(* IEC 61131-3 sources: volt/packages/volt-lsp-iec/test-corpus/pro2193/Device/Plc Logic/Application/03 Hardware Units/32 BFU/32.10 - Fanuc/Project, 1 file *)

(* ---- FanucUnitFB.pou ---- *)
{attribute 'symbol' := 'none'}
FUNCTION_BLOCK FanucUnitFB
EXTENDS FanucUnitBaseFB
VAR_INPUT
END_VAR
VAR_OUTPUT
END_VAR
VAR_IN_OUT
	DataProject					: FanucUnit_Data;
END_VAR
VAR
END_VAR

%LANGUAGE ST
SUPER^(
	Data			:= Data,
	GripperStatus	:= GripperStatus
);

END_FUNCTION_BLOCK
